Staubli VAL3: MotionAddon.pjx

--- MotionAddon.pjx ---
Parameters version=s7.9.1 stackSize=5000 millimeterUnit=true
Program file=equival_Trsf.pgx
Program file=externalFrc.pgx
Program file=getCycleTime.pgx
Program file=getPosFbk.pgx
Program file=motionState.pgx
Program file=readMe.pgx
Program file=start.pgx
Program file=stop.pgx
Data file=MotionAddon.dtx

--- MotionAddon.dtx ---
mdesc mNomSpeed
trsf tTransformation = {rx=90}
num nXaxis
num nYaxis
num nZaxis
num nAngle
trsf trNew
num nSetAngle
num nSetXaxis
num nSetYaxis
num nSetZaxis
tool tTool = {fatherId=flange[0], ioLink=valve1}
pointRx pFbk = {fatherId=world[0]}
jointRx jFbk
num nCycleTime
num nMotState
num nMotStBit[17]
trsf trWorldExtFrc
trsf trTCPExtFrc

--- start.pgx ---
program start()
begin
  //
  userPage()
  cls()
  gotoxy(1,1)
  put("F1->等效轴与Trsf转换")
  gotoxy(1,2)
  put("F2->获取反馈位置")
  gotoxy(1,3)
  put("F3->计算外力")
  gotoxy(1,4)
  put("F4->系统周期")
  gotoxy(1,5)
  put("F5->机器人运动状态")
  while true

    switch getKey()
      case 271
        call equival_Trsf()
      break
      case 272
        call getPosFbk()
      break
      case 273
        call externalFrc()
      break
      case 274
        call getCycleTime()
      break
      case 275
        call motionState()
      break
    endSwitch
    delay(0)
  endWhile
end

--- equival_Trsf.pgx ---
program equival_Trsf()
begin
  //等效轴变换与Trsf变量之间的转换。


  cls()
  //从一个trsf中获取变换转角
  nAngle=$rotAngle(tTransformation)
  //
  gotoxy(0,0)
  put("变换：")
  gotoxy(0,1)
  put("x:"+toString("7.3",tTransformation.x))
  gotoxy(0,2)
  put("y:"+toString("7.3",tTransformation.y))
  gotoxy(0,3)
  put("z:"+toString("7.3",tTransformation.z))
  gotoxy(15,1)
  put("rx:"+toString("7.3",tTransformation.rx))
  gotoxy(15,2)
  put("ry:"+toString("7.3",tTransformation.ry))
  gotoxy(15,3)
  put("rz:"+toString("7.3",tTransformation.rz))
  gotoxy(0,4)
  put("通用转角："+toString("5.2",nAngle))

  //返回通用轴和转角
  nAngle=$getRot(tTransformation,nXaxis,nYaxis,nZaxis)
  gotoxy(0,6)
  put("通用转轴："+toString("5.3",nXaxis)+","+toString("5.3",nYaxis)+","+toString("5.3",nZaxis))
  gotoxy(0,7)
  put("通用转角："+toString("5.2",nAngle))

  //把通用轴和转角转换成标准变换矩阵
  if nSetXaxis*nSetXaxis+nSetYaxis*nSetYaxis+nSetZaxis*nSetZaxis>0
    trNew=$setRot(nSetAngle,nSetXaxis,nSetYaxis,nSetZaxis)
    gotoxy(0,8)
    put("通用转轴："+toString("5.3",nSetXaxis)+","+toString("5.3",nSetYaxis)+","+toString("5.3",nSetZaxis))
    gotoxy(0,9)
    put("通用转角："+toString("5.2",nSetAngle))
    //
    gotoxy(0,10)
    put("得到的变换：")
    gotoxy(0,11)
    put("x:"+toString("7.3",trNew.x))
    gotoxy(0,12)
    put("y:"+toString("7.3",trNew.y))
    gotoxy(0,13)
    put("z:"+toString("7.3",trNew.z))
    gotoxy(15,11)
    put("rx:"+toString("7.3",trNew.rx))
    gotoxy(15,12)
    put("ry:"+toString("7.3",trNew.ry))
    gotoxy(15,13)
    put("rz:"+toString("7.3",trNew.rz))
  else
    gotoxy(0,8)
    put("通用转轴："+"错误")
    gotoxy(0,9)
    put("通用转角："+toString("5.2",nSetAngle))
    //
    gotoxy(0,10)
    put("得到的变换：")
    gotoxy(0,11)
    put("x:"+"-")
    gotoxy(0,12)
    put("y:"+"-")
    gotoxy(0,13)
    put("z:"+"-")
    gotoxy(15,11)
    put("rx:"+"-")
    gotoxy(15,12)
    put("ry:"+"-")
    gotoxy(15,13)
    put("rz:"+"-")
  endIf
end

--- externalFrc.pgx ---
program externalFrc()
  local joint l_jPos
  local num l_nCurJntTorq[6]
  local num l_nJntVel[6]
  local num l_nJntVelPrev[6]
  local num l_nJntAccel[6]
  local num l_nCycleTime
  local num l_nTheoJntTorq[6]
  local num l_nJntExtTorq[6]
  local num l_nWorldExtFrc[6]
  local trsf l_trWorldOvrFrc
  local point l_pHere
  local num l_ni
begin
  cls()
  //获取系统周期
  l_nCycleTime=$getCycleTime()

  //每一个系统周期计算一次外部力
  while true
    //读取反馈位置
    l_jPos=$getJntFbk()
    //读取关节力矩
    getJointForce(l_nCurJntTorq)
    //读取关节速度
    $getJntSpeedFbk(l_nJntVel)
    //计算关节加速度
    for l_ni=0 to 5
      l_nJntAccel[l_ni]=(l_nJntVel[l_ni]-l_nJntVelPrev[l_ni])/l_nCycleTime
      l_nJntVelPrev[l_ni]=l_nJntVel[l_ni]
    endFor
    //根据重力和马达特性计算理论关节力矩
    $computeJntFrc(l_jPos,l_nJntVel,l_nJntAccel,l_nTheoJntTorq)

    //计算关节力矩实际值与理论值的偏差
    for l_ni=0 to 5
      l_nJntExtTorq[l_ni]=l_nCurJntTorq[l_ni]-l_nTheoJntTorq[l_ni]
    endFor
    //计算世界坐标下TCP处的力或力矩
    $externalForce(l_jPos,tTool,l_nJntExtTorq,l_nWorldExtFrc)

    //这里不考虑力矩,world下的外力表示：x,y,z分量
    trWorldExtFrc.x=l_nWorldExtFrc[0]
    trWorldExtFrc.y=l_nWorldExtFrc[1]
    trWorldExtFrc.z=l_nWorldExtFrc[2]
    //
    //
    //把力换算到TCP坐标系下
    //获取TCP位置
    l_pHere=here(tTool,world)
    //保留旋转量
    l_pHere.trsf.x=0
    l_pHere.trsf.y=0
    l_pHere.trsf.z=0
    //保留力：x，y，z分量
    l_trWorldOvrFrc.x=l_nWorldExtFrc[0]
    l_trWorldOvrFrc.y=l_nWorldExtFrc[1]
    l_trWorldOvrFrc.z=l_nWorldExtFrc[2]
    //
    trTCPExtFrc=l_pHere.trsf*l_trWorldOvrFrc

    //屏幕输出(实际)不需要
    //
    gotoxy(1,0)
    put("机器人受到的外力：")
    gotoxy(1,2)
    put("World下的表示:")
    gotoxy(1,3)
    put("x:"+toString("8.3",trWorldExtFrc.x))
    gotoxy(1,4)
    put("y:"+toString("8.3",trWorldExtFrc.y))
    gotoxy(1,5)
    put("z:"+toString("8.3",trWorldExtFrc.z))
    //TCP处
    gotoxy(1,7)
    put("TCP下的表示:")
    gotoxy(1,8)
    put("x:"+toString("8.3",trTCPExtFrc.x))
    gotoxy(1,8)
    put("y:"+toString("8.3",trTCPExtFrc.y))
    gotoxy(1,8)
    put("z:"+toString("8.3",trTCPExtFrc.z))
    delay(0)
  endWhile
end

--- getCycleTime.pgx ---
program getCycleTime()
begin
  //
  cls()
  //
  nCycleTime=$getCycleTime()
  //
  gotoxy(1,0)
  put("当前系统周期(s)："+toString("4.3",nCycleTime))
end

--- getPosFbk.pgx ---
program getPosFbk()
begin
  cls()
  //point
  pFbk=$getPosFbk(tTool,world)
  gotoxy(1,0)
  put("当前笛卡尔反馈位置:")
  gotoxy(1,1)
  put("x:"+toString("8.3",pFbk.trsf.x))
  gotoxy(1,2)
  put("y:"+toString("8.3",pFbk.trsf.y))
  gotoxy(1,3)
  put("z:"+toString("8.3",pFbk.trsf.z))
  gotoxy(20,1)
  put("rx:"+toString("8.3",pFbk.trsf.rx))
  gotoxy(20,2)
  put("ry:"+toString("8.3",pFbk.trsf.ry))
  gotoxy(20,3)
  put("rz:"+toString("8.3",pFbk.trsf.rz))
  //joint
  jFbk=$getJntFbk()
  gotoxy(1,5)
  put("当前关节反馈位置:")
  gotoxy(1,6)
  put("j1:"+toString("8.3",jFbk.j1))
  gotoxy(1,7)
  put("j2:"+toString("8.3",jFbk.j2))
  gotoxy(1,8)
  put("j3:"+toString("8.3",jFbk.j3))
  gotoxy(20,6)
  put("j4:"+toString("8.3",jFbk.j4))
  gotoxy(20,7)
  put("j5:"+toString("8.3",jFbk.j5))
  gotoxy(20,8)
  put("j6:"+toString("8.3",jFbk.j6))
end

--- motionState.pgx ---
program motionState()
  local num l_ni
  local num l_nMask
  local string l_sTemp
begin
  //
  cls()
  //
  nMotState=$motionState()
  //
  //检测返回数值的二进制数哪些位上是“1”
  //根据函数说明：0-14和15-29取值相同，30,31位还计算
  for l_ni=0 to 14
    l_nMask=power(2,l_ni)
    if bAnd(nMotState,l_nMask)==l_nMask
      nMotStBit[l_ni]=1
    endIf
  endFor
  //
  for l_ni=30 to 31
    l_nMask=power(2,l_ni)
    if bAnd(nMotState,l_nMask)==l_nMask
      nMotStBit[l_ni-15]=1
    endIf
  endFor
  //
  //通过对nMotStBit的判断并查看说明可以等到信息。
  gotoxy(1,0)
  put("当前运动状态:")
  for l_ni=0 to 16
    l_sTemp=l_sTemp+toString("",nMotStBit[l_ni])
  endFor
  gotoxy(1,1)
  put(l_sTemp)

end

--- readMe.pgx ---
public program readMe()
begin
  //
  //
  //
end
